# B&R Automation Studio project AsProject
Automation Studio 4.11.4.55 SP; Starter Automation Studio project.

## Configuration StarterConfig

CPU 5PC900.TS17-04, AutomationRuntime C4.90, Build 6.3.0, Vc V4.72.0

### Task classes (Cpu.sw)
```
Cyclic#1 (cycle 2000 us, tolerance 0 us):
  FirstInitP <- Infrastructure.FirstInitProg.prg
  demo <- demo.prg
  demoGlobal <- demoGlobal.prg
  Page <- Page.prg
Cyclic#8:
  LuxProg <- Lux.LuxProg.prg
Binaries: udbdef, TCData, FWRules, ashwd, ashwac, User, sysconf, asfw, arconfig, iomap, Role
Libraries: ArEventLog, AsARCfg, AsArLog, AsArProf, AsBrMath, AsBrStr, AsDb, AsEPL, AsGuard, AsHttp, AsIO, AsIOAcc, AsIODiag, AsIOTime, AsMem, AsSafety, AsSem, AsTCP, astime, AsUDP, AsUSB, AsXml, AsZip, brsystem, Convert, DataObj, dvframe, FileIO, MTBasics, MTLookUp, MTTypes, LoopConR, operator, runtime, standard, sys_lib, AsBrWStr, omjson, vartools, databuffer, tcpcomm, websocket, persist, csvfilelib, fiowrap, errorlib, hmitools, ringbuflib, stringext, logthat
```

### Hardware
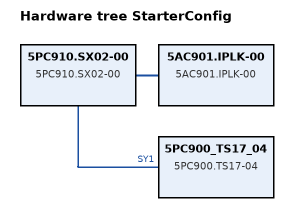
```
5AC901.IPLK-00 : 5AC901.IPLK-00 v1.7.1.0  [SS -> 5PC910.SX02-00.SS2]
  Connector IF1:
    DNAConfiguration = manual
5PC900_TS17_04 : 5PC900.TS17-04 v2.1.0.0  [SY -> 5PC910.SX02-00.SY1]
  ConfigurationID = Starter_StarterConfig
  UserPartitionSize = 300
  Simulation = 1
  UserRamDevice = PCI.2.IPLK.SRAM
  UserRamSize = 500000
  RemMemDevice = PCI.2.IPLK.SRAM
  RemMemSize = 120000
  PermanentPvSize = 10000
  RemanentGlobalPvSize = 105000
  VolatileGlobalPvSize = 1000000
  TimerDeviceType = EPLX2X
  TimerDevice = 5AC901.IPLK-00.IF1
  IdleTaskClass = 3
  TaskClassIdleTime = 8000
  Cyclic1Duration = 2000
  Cyclic1Tolerance = 0
  Cyclic2Duration = 10000
  Cyclic3Duration = 20000
  Cyclic3Tolerance = 40000
  TimeZone = 25
  FtpUser1
  FtpUsername1 = dev
  FtpUserPassword1 = NYwXHzz4INzZvtlFBMOTmjZqrH4JRkY3Uye1yrmlNSg=  // dev
  FtpUserSalt1 = s9/ksXy4
  FTPAccessRight1 = 0
  FTPdevice1 = ALL
  SdmColor = colorRGB
5PC910.SX02-00 : 5PC910.SX02-00 v2.1.0.0
  Connector IF1:
    AssignedOperatingSystem = ARemb
  Connector IF3:
    AssignedOperatingSystem = ARemb
    ActivateDevice = 1
  Connector IF4:
    AssignedOperatingSystem = ARemb
    ActivateDevice = 1
  Connector IF5:
    AssignedOperatingSystem = ARemb
  Connector IF6:
    AssignedOperatingSystem = ARemb
  Connector IF7:
    AssignedOperatingSystem = ARemb
  Connector IF8:
    AssignedOperatingSystem = ARemb
  Connector IF9:
    AssignedOperatingSystem = ARemb
```

- Physical/StarterConfig/5PC900_TS17_04/IoMap.iom: same as Physical/StarterConfig/5PC900_TS17_04/Cpu.per
- Physical/StarterConfig/5PC900_TS17_04/PvMap.vvm: same as Physical/StarterConfig/5PC900_TS17_04/Cpu.per
## Logical view

Binary libraries used (declarations not repeated): ArEventLog, AsARCfg, AsArLog, AsArProf, AsBrMath, AsBrStr, AsDb, AsEPL, AsGuard, AsHttp, AsIO, AsIOAcc, AsIODiag, AsIOTime, AsMem, AsSafety, AsSem, astime, AsTCP, AsUDP, AsUSB, AsXml, AsZip, brsystem, Convert, DataObj, dvframe, FileIO, LoopConR 4.10.2, MTBasics 5.12.0, MTLookUp 5.12.0, MTTypes 1.03.4, operator, runtime, standard, sys_lib, AsBrWStr, omjson 1.04.0, vartools 0.11.3, databuffer 0.01.1, tcpcomm 0.10.0, websocket 0.02.0, csvfilelib 1.02.2, fiowrap 0.09.1, errorlib 0.23.3, hmitools 0.11.4, ringbuflib 0.02.4, stringext 0.14.4, logthat 0.05.1, persist 0.00.7

### Global.var - Global variables
```iecst
VAR
	test : TestStruct;
END_VAR
```

### Types.typ - Local data types
```iecst
TYPE
	TestStruct : 	STRUCT
		command : BOOL;
		slider : REAL;
		random : REAL;
		struct2 : TestStruct1;
		struct3 : TestStruct1;
		struct1 : TestStruct1;
		myvalue : TestStruct3;
	END_STRUCT;
	TestStruct1 : 	STRUCT
		struct1 : TestStruct2;
		struct2 : TestStruct2;
	END_STRUCT;
	TestStruct2 : 	STRUCT
		member : BOOL;
		member1 : INT;
		member2 : DINT;
		member3 : STRING[80];
	END_STRUCT;
	TestStruct3 : 	STRUCT
		x : REAL;
	END_STRUCT;
END_TYPE
```

### Package Logical/Libraries - Global libraries

### Lux.var
```iecst
VAR
	gWSTimeout : BOOL;
	jsonWebSocketServer_0 : jsonWebSocketServer;
END_VAR
```

### Program Logical/Lux/LuxProg (IEC)

#### Main.st - Cyclic code
```iecst
// This program serves variables to web applications via WebSockets and
// a JSON interface

PROGRAM _INIT

    // pCache is required
	jsonWebSocketServer_0.pCacheArray := ADR(jsonCache);
	jsonWebSocketServer_0.maxClients := MAX_CLIENTS;

	// Note: ServerIP, ServerPort, BufferSize, and MaxIterations are optional and not set
	jsonWebSocketServer_0.BufferSize := 200000;

	// Call jsonWebSocketServer once in the INIT routine to allocate internal memory
	jsonWebSocketServer_0();

END_PROGRAM

PROGRAM _CYCLIC

	// Call jsonWebSocketServer cyclically to serve variables
	jsonWebSocketServer_0();

	IF NOT gSimulation THEN
		gWSTimeout := FALSE;
		FOR i:=0 TO JSON_MAI_CLIENTS DO
			// On any client disconnect
			IF oldClientInfo[i].Connected AND NOT jsonWebSocketServer_0.ClientInfo[i].Connected THEN
				gWSTimeout := TRUE;
			END_IF
		END_FOR
		oldClientInfo := jsonWebSocketServer_0.ClientInfo;
	END_IF

END_PROGRAM
```

#### Variables.var - Local variables
```iecst
VAR
	i : UINT;
	jsonCache : ARRAY[0..MAI_CLIENTS] OF jsonCache_typ;
END_VAR
VAR CONSTANT
	MAI_CLIENTS : USINT := MAX_CLIENTS-1;
	MAX_CLIENTS : USINT := 2;
END_VAR
VAR
	oldClientInfo : ARRAY[0..JSON_MAI_CLIENTS] OF jsonWSS_client_info_typ;
END_VAR
```

### Program Logical/Infrastructure/FirstInitProg (ANSIC)

#### FirstInitProgInit.c - Initialization code
```c
/*
 * File: FirstInitProgInit.c
 * Copyright (c) 2023 Loupe
 * https://loupe.team
 *
 * This file is part of FirstInitProg, licensed under the MIT License.
 */

#include <bur/plctypes.h>

#ifdef _DEFAULT_INCLUDES
#include <AsDefault.h>
#endif

#include <string.h>

void _INIT FirstInitProgInit(void)
{
	// Set gTransfer to be whether or not FirstInit cyclic has ran
	gTransfer.transfer = gTransfer.cyclic;

	// Check to see if this is a new transfer or FirstInit cyclic has ran
	//if( strcmp(_buildDate, buildDate) != 0 || gTransfer.transfer){
	//	gTransfer.bootAfterTransfer = !gTransfer.transfer;
	//}

	// Update build date
	//if(!gTransfer.transfer){
	//	strcpy(_buildDate, buildDate);
	//}
	// Check for simulation
	// This is a DevLink using a Windows share which is not supported by ARsim
	// We use this instead of Diag function to support older CPU's
	simCheckDevLink.enable = 1;
	simCheckDevLink.pDevice = (UDINT)&("SimCheck");
	simCheckDevLink.pParam = (UDINT)&("/SIP=127.0.0.1 /PROTOCOL=cifs /SHARE=testfolder /USER=max /PASSWORD=passw");

	DevLink(&simCheckDevLink);

	if (simCheckDevLink.status == ERR_NOTIMPLEMENTED) {
		gSimulation = 1;
	}

	// Initialize User Loggers
	createLogInit("Errors", 1000000, arEVENTLOG_PERSISTENCE_VOLATILE);
	createLogInit("Files", 1000000, arEVENTLOG_PERSISTENCE_VOLATILE);
	createLogInit("Application", 1000000, arEVENTLOG_PERSISTENCE_VOLATILE);

	// Initialize error collector
	//ErrorCollectorFn_Init(&gErrorCollector);

	// Link file devices
	//-------------------------------------------------------

	// This is NOT done in the CPU configuration because when using CPU simulation
	// you cannot have separate file devices for simulation mode,
	// and you cannot unlink devices that were entered in the CPU configuration

	// Set up file device names
	strcpy(fileDevice[0], "CF_User");
	strcpy(fileDevice[1], "CNC_PrgDir");
	strcpy(fileDevice[2], "Recipes");
	strcpy(fileDevice[3], "permBackup");

	// Set up file device paths
	if (gSimulation) {
		strcpy(directory[0], "C:\\ARSimUser\\Sandbox");
		strcpy(directory[1], "C:\\ARSimUser\\Sandbox\\CNC");
		strcpy(directory[2], "C:\\ARSimUser\\Sandbox\\Recipes");
		strcpy(directory[3], "C:\\ARSimUser\\Sandbox\\PermData");
	} else {
		// TODO: This won't work (nicely) with ARwin
		strcpy(directory[0], "F:\\");
		strcpy(directory[1], "F:\\CNC");
		strcpy(directory[2], "F:\\Recipes");
		strcpy(directory[3], "F:\\PermData");
	}

	// Link file devices
	for (i = 0; i < NUM_FILEDEVICES; i++) {

		strcpy(parameters[i], "/DEVICE=");
		strcat(parameters[i], directory[i]);

		fileDeviceDevLink[i].enable = 1;
		fileDeviceDevLink[i].pDevice = (UDINT)&(fileDevice[i]);
		fileDeviceDevLink[i].pParam = (UDINT)&(parameters[i]);

		DevLink(&fileDeviceDevLink[i]);

		//if (fileDeviceDevLink[i].status != 0)
		//	errcolAddError((UDINT)"File Devices", (UDINT)"Error linking file device", fileDeviceDevLink[i].status, 0, &gErrorCollector);

	}

	// Initialize Persisters
	//-------------------------------------------------------

	#ifdef NUM_PERSISTERS
	// Reset the data if we need to
	if (gTransfer.bootAfterTransfer || gTransfer.transfer) {
		// Reset all data valids to false
		for (i = 0; i < NUM_PERSISTERS; i++) {
			gDataValid[i] = 0;
		}
	}

	// Working variables

	// Machine configuration
	varGetVariableList((UDINT)"Configuration", (UDINT)&(gPersister[PERM_CONFIGURATION].IN.WorkingVariableList));

	// Home data
	strcpy(gPersister[PERM_HOME_DATA].IN.WorkingVariableList[0],"gEndlessPosition");

	// Axis pars
	// TODO: I think we should move away from gMotorBasic inside persisters and towards local Configuration variables
	#ifdef NUM_MOTOR 	// Only execute this loop if NUM_MOTOR is defined by ServoControl
	for (i = 0; i < NUM_MOTOR; i++) {
		brsitoa(i, (UDINT)indexString);
		strcpy(axisString, "gMotorBasic");
		appendArrayIndex(i, (UDINT)axisString);
		strcat(axisString, ".IN.PAR");
		if (i <= PERSIST_MAI_VARLIST) {
			strcpy(gPersister[PERM_AXIS_PARS].IN.WorkingVariableList[i], axisString);
		} else {
			errcolAddError((UDINT)"Perm Data", (UDINT)"Too many axes for one persister.", 0, 0, &gErrorCollector);
			break;
		}
	}
	#endif

	// Permanent variables
	gPersister[PERM_CONFIGURATION].IN.pPersistentVariable = (UDINT)&gPermConfiguration;
	gPersister[PERM_CONFIGURATION].IN.sizeofPersistentVariable = sizeof(gPermConfiguration);

	gPersister[PERM_HOME_DATA].IN.pPersistentVariable = (UDINT)&gPermHomeData;
	gPersister[PERM_HOME_DATA].IN.sizeofPersistentVariable = sizeof(gPermHomeData);

	gPersister[PERM_AXIS_PARS].IN.pPersistentVariable = (UDINT)&gPermAxisPars;
	gPersister[PERM_AXIS_PARS].IN.sizeofPersistentVariable = sizeof(gPermAxisPars);

	gPersister[PERM_AXIS_CFG].IN.pPersistentVariable = (UDINT)&gPermAxisCfgs;
	gPersister[PERM_AXIS_CFG].IN.sizeofPersistentVariable = sizeof(gPermAxisCfgs);

	// DataValid and PersistFn_Init()
	for(i = 0; i < NUM_PERSISTERS; i++){
		gPersister[i].IN.pDataValid = (UDINT)&gDataValid[i];
		PersistFn_Init(&gPersister[i]);
		if(gPersister[i].OUT.STAT.Error){
			errcolAddError((UDINT)"Perm Data", (UDINT)gPersister[i].OUT.STAT.ErrorString, gPersister[i].OUT.STAT.ErrorID, 0, &gErrorCollector);
		}
	}

	// Initialize persister CSV backups
	errcolAddSourceByName((UDINT)"Machine configuration backup", (UDINT)"gPermBackup[0]", &gErrorCollector);
	errcolAddSourceByName((UDINT)"Home data backup", (UDINT)"gPermBackup[1]", &gErrorCollector);
	errcolAddSourceByName((UDINT)"Axis pars backup", (UDINT)"gPermBackup[2]", &gErrorCollector);
	errcolAddSourceByName((UDINT)"Axis cfg backup", (UDINT)"gPermBackup[3]", &gErrorCollector);

	strcpy(gPermBackup[PERM_CONFIGURATION].IN.PAR.FileName, "configuration.csv");
	strcpy(gPermBackup[PERM_HOME_DATA].IN.PAR.FileName, "homeData.csv");
	strcpy(gPermBackup[PERM_AXIS_PARS].IN.PAR.FileName, "axisPars.csv");
	strcpy(gPermBackup[PERM_AXIS_CFG].IN.PAR.FileName, "axisCfg.csv");

	for( i = 0; i < NUM_PERSISTERS; i++){

		strcpy(gPermBackup[i].IN.PAR.FileDevice, "permBackup");
		memcpy(&gPermBackup[i].IN.PAR.VariableList, &gPersister[i].IN.WorkingVariableList, sizeof(gPermBackup[i].IN.PAR.VariableList) );

		strcpy(gPermBackup[i].IN.CFG.LogFileName, ".csvlogPermBackup");
		brsitoa(i, (UDINT)indexString);
		strcat(gPermBackup[i].IN.CFG.LogFileName, indexString);

		CSVFn_Init(&(gPermBackup[i]));

		if (!gDataValid[i]) {
			CSVOpenFile_Init(&gPermBackup[i]);
			if (!gPermBackup[i].OUT.STAT.Error) {
				gDataValid[i] = 1;
				errcolAddError((UDINT)"Data restored", (UDINT)&(gPermBackup[i].IN.PAR.FileName), 0, 0, &gErrorCollector);
			}
		}

	} // loop through permbackup

	// Load configuration.csv every startup
	//CSVOpenFile_Init(&gPermBackup[PERM_CONFIGURATION]);

	#endif

} // _INIT
```

#### FirstInitProgCyclic.c - Cyclic code
```c
/*
 * File: FirstInitProgCyclic.c
 * Copyright (c) 2023 Loupe
 * https://loupe.team
 *
 * This file is part of FirstInitProg, licensed under the MIT License.
 */

#include <bur/plctypes.h>

#ifdef _DEFAULT_INCLUDES
	#include <AsDefault.h>
#endif

void _CYCLIC FirstInitProgCyclic(void)
{
	// Set our cyclic bit to true once FirstInit cyclic runs
	// This is to tell the init routine if the cyclic has ran
	gTransfer.cyclic = 1;

	// DO NOT ADD ANY "OTHER" CYCLIC CODE HERE! //
	//if( strcmp(_buildDate, buildDate) != 0 ){
	//	gTransfer.transfer = 1;
	//}
}
```

#### FirstInitProg.var - Local variables
```iecst
(********************************************************************
 * File: FirstInitProg.var
 * Copyright (c) 2023 Loupe
 * https://loupe.team
 *
 * This file is part of FirstInitProg, licensed under the MIT License.
 ********************************************************************)
VAR CONSTANT
	NUM_FILEDEVICES : USINT := 4;
	MAI_FILEDEVICES : USINT := NUM_FILEDEVICES-1;
END_VAR
VAR
	simCheckDevLink : DevLink := (0);
	fileDeviceDevLink : ARRAY[0..MAI_FILEDEVICES] OF DevLink := [4(0)];
	fileDevice : ARRAY[0..MAI_FILEDEVICES] OF STRING[20] := [4('')];
	directory : ARRAY[0..MAI_FILEDEVICES] OF STRING[320] := [4('')];
	parameters : ARRAY[0..MAI_FILEDEVICES] OF STRING[320] := [4('')];
	i : DINT := 0;
	indexString : STRING[320] := '';
	axisString : STRING[320] := '';
END_VAR
VAR RETAIN
	_buildDate : STRING[80];
END_VAR
```

### Infrastructure.typ
```iecst
(********************************************************************
 * File: Infrastructure.typ
 * Copyright (c) 2023 Loupe
 * https://loupe.team
 *
 * This file is part of FirstInitProg, licensed under the MIT License.
 ********************************************************************)
TYPE
	Transfer_typ : 	STRUCT
		cyclic : BOOL;
		transfer : BOOL;
		bootAfterTransfer : BOOL;
	END_STRUCT;
END_TYPE
```

### Infrastructure.var
```iecst
(********************************************************************
 * File: Infrastructure.var
 * Copyright (c) 2023 Loupe
 * https://loupe.team
 *
 * This file is part of FirstInitProg, licensed under the MIT License.
 ********************************************************************)
(*Persisters to handle memory management*)
VAR
	gSimulation : BOOL;
END_VAR
(*Permanent memory chunks*)
VAR RETAIN
	gPermHomeData : ARRAY[0..999] OF USINT;
END_VAR
(*Variables to handle transfers*)
VAR
	gTransfer : Transfer_typ;
END_VAR
```

### Program Logical/demo (IEC)

#### Main.st - Init, cyclic, exit code
```iecst
PROGRAM _INIT
	test;

END_PROGRAM

PROGRAM _CYCLIC
	(* Insert code here *)

END_PROGRAM

PROGRAM _EXIT
	(* Insert code here *)

END_PROGRAM
```

#### Variables.var - Local variables
```iecst
VAR
	test : TestStruct;
END_VAR
```

### Program Logical/demoGlobal (IEC)

#### Main.st - Init, cyclic, exit code
```iecst
PROGRAM _INIT
	test;

END_PROGRAM

PROGRAM _CYCLIC
	(* Insert code here *)

END_PROGRAM

PROGRAM _EXIT
	(* Insert code here *)

END_PROGRAM
```

### Program Logical/Page (IEC)

#### Cyclic.st - Cyclic code
```iecst
PROGRAM _CYCLIC
	(* Insert code here *)

END_PROGRAM
```

#### Init.st - Init code
```iecst
PROGRAM _INIT
	(* Insert code here *)

END_PROGRAM
```

#### Exit.st - Exit code
```iecst
PROGRAM _EXIT
	(* Insert code here *)

END_PROGRAM
```

#### Types.typ - Local data types
```iecst
TYPE
	myVar_typ : 	STRUCT
		in : myVar_in_typ;
		out : myVar_out_typ;
	END_STRUCT;
	myVar_in_typ : 	STRUCT
		command : USINT;
	END_STRUCT;
	myVar_out_typ : 	STRUCT
		state : USINT;
	END_STRUCT;
END_TYPE
```

#### Variables.var - Local variables
```iecst
VAR
	MyVar : myVar_typ;
END_VAR
```
